FUNCTION_BLOCK TIMER
VAR_INPUT
	In1: BOOL;
END_VAR
VAR_OUTPUT
	out1: BOOL;
END_VAR
VAR
	Timer1: TON;
	ontValue: TIME;
END_VAR

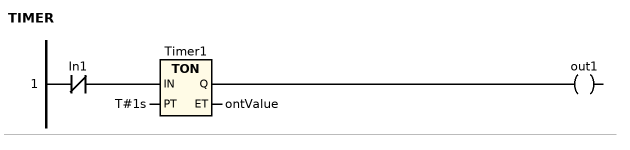
// NETWORK 1
Timer1(IN := NOT In1, PT := T#1s, ET => ontValue); // TON
out1 := Timer1.Q;

END_FUNCTION_BLOCK

(* stored: Version 1.1.0.1, ProductVersion 3.1.4024.15
   POU TIMER: Id {dc118c13-cd4e-4ae7-859f-76d6815d496b}, SpecialFunc None *)
